(* IEC 61131-3 sources: com.logicals.lc3.webinar/logicals_Lib_Webinar/logicals_Webinar_Basic_Lib/logicals_Lib/src_FB_FBD/Convert, 5 files *)

(* ---- FB_lc_ByteNotNull_FBD.iecfbd ---- *)
NAMESPACE com.logicals.Basic.Convert
FUNCTION_BLOCK FB_lc_ByteNotNull_FBD
  {
    width := 170;
    minWidth := 160;
    maxWidth := 160;
    height := 198;
    minHeight := 198;
    maxHeight := 198;
  }

  VAR_INPUT
    vib_Byte9 : BYTE := 95;
    vib_Byte8 : BYTE := 95;
    vib_Byte7 : BYTE := 95;
    vib_Byte6 : BYTE := 95;
    vib_Byte5 : BYTE := 95;
    vib_Byte4 : BYTE := 95;
    vib_Byte3 : BYTE := 95;
    vib_Byte2 : BYTE := 95;
    vib_Byte1 : BYTE := 95;
    vib_Byte0 : BYTE := 95;
  END_VAR
  VAR_OUTPUT
    vob_Byte9 : BYTE := 95;
    vob_Byte8 : BYTE := 95;
    vob_Byte7 : BYTE := 95;
    vob_Byte6 : BYTE := 95;
    vob_Byte5 : BYTE := 95;
    vob_Byte4 : BYTE := 95;
    vob_Byte3 : BYTE := 95;
    vob_Byte2 : BYTE := 95;
    vob_Byte1 : BYTE := 95;
    vob_Byte0 : BYTE := 95;
  END_VAR

  (*

    // Network 1:
    EQ(IN1 := vib_Byte0, IN2 := 0, EQ => @C(161).EQ);
    SEL(G := @C(161).EQ, IN0 := vib_Byte0, IN1 := 95, SEL => vob_Byte0);

    // Network 2:
    EQ(IN1 := vib_Byte1, IN2 := 0, EQ => @C(160).EQ);
    SEL(G := @C(160).EQ, IN0 := vib_Byte1, IN1 := 95, SEL => vob_Byte1);

    // Network 3:
    EQ(IN1 := vib_Byte2, IN2 := 0, EQ => @C(164).EQ);
    SEL(G := @C(164).EQ, IN0 := vib_Byte2, IN1 := 95, SEL => vob_Byte2);

    // Network 4:
    EQ(IN1 := vib_Byte3, IN2 := 0, EQ => @C(162).EQ);
    SEL(G := @C(162).EQ, IN0 := vib_Byte3, IN1 := 95, SEL => vob_Byte3);

    // Network 5:
    EQ(IN1 := vib_Byte4, IN2 := 0, EQ => @C(166).EQ);
    SEL(G := @C(166).EQ, IN0 := vib_Byte4, IN1 := 95, SEL => vob_Byte4);

    // Network 6:
    EQ(IN1 := vib_Byte5, IN2 := 0, EQ => @C(169).EQ);
    SEL(G := @C(169).EQ, IN0 := vib_Byte5, IN1 := 95, SEL => vob_Byte5);

    // Network 7:
    EQ(IN1 := vib_Byte6, IN2 := 0, EQ => @C(165).EQ);
    SEL(G := @C(165).EQ, IN0 := vib_Byte6, IN1 := 95, SEL => vob_Byte6);

    // Network 8:
    EQ(IN1 := vib_Byte7, IN2 := 0, EQ => @C(168).EQ);
    SEL(G := @C(168).EQ, IN0 := vib_Byte7, IN1 := 95, SEL => vob_Byte7);

    // Network 9:
    EQ(IN1 := vib_Byte8, IN2 := 0, EQ => @C(163).EQ);
    SEL(G := @C(163).EQ, IN0 := vib_Byte8, IN1 := 95, SEL => vob_Byte8);

    // Network 10:
    EQ(IN1 := vib_Byte9, IN2 := 0, EQ => @C(167).EQ);
    SEL(G := @C(167).EQ, IN0 := vib_Byte9, IN1 := 95, SEL => vob_Byte9);

  *)

  @C(118) : @F(SEL), @R(810.0, 820.0, 120.0, 58.0), BYTE, @I(@N(G), @L(9.5)), @I(@N(IN0), @L(29.5)), @I(@N(IN1), @L(49.5)), @O(@N(SEL), @R(9.5));
  @C(150) : @F(SEL), @R(810.0, 730.0, 120.0, 58.0), BYTE, @I(@N(G), @L(9.5)), @I(@N(IN0), @L(29.5)), @I(@N(IN1), @L(49.5)), @O(@N(SEL), @R(9.5));
  @C(163) : @F(EQ), @R(540.0, 730.0, 40.0, 38.0), BYTE, @I(@N(IN1), @L(9.5)), @I(@N(IN2), @L(29.5)), @O(@N(EQ), @R(9.5));
  @C(167) : @F(EQ), @R(540.0, 820.0, 40.0, 38.0), BYTE, @I(@N(IN1), @L(9.5)), @I(@N(IN2), @L(29.5)), @O(@N(EQ), @R(9.5));
  @C(143) : @F(SEL), @R(810.0, 640.0, 120.0, 58.0), BYTE, @I(@N(G), @L(9.5)), @I(@N(IN0), @L(29.5)), @I(@N(IN1), @L(49.5)), @O(@N(SEL), @R(9.5));
  @C(168) : @F(EQ), @R(540.0, 640.0, 40.0, 38.0), BYTE, @I(@N(IN1), @L(9.5)), @I(@N(IN2), @L(29.5)), @O(@N(EQ), @R(9.5));
  @C(148) : @F(SEL), @R(810.0, 550.0, 120.0, 58.0), BYTE, @I(@N(G), @L(9.5)), @I(@N(IN0), @L(29.5)), @I(@N(IN1), @L(49.5)), @O(@N(SEL), @R(9.5));
  @C(165) : @F(EQ), @R(540.0, 550.0, 40.0, 38.0), BYTE, @I(@N(IN1), @L(9.5)), @I(@N(IN2), @L(29.5)), @O(@N(EQ), @R(9.5));
  @C(156) : @F(SEL), @R(810.0, 460.0, 120.0, 58.0), BYTE, @I(@N(G), @L(9.5)), @I(@N(IN0), @L(29.5)), @I(@N(IN1), @L(49.5)), @O(@N(SEL), @R(9.5));
  @C(169) : @F(EQ), @R(540.0, 460.0, 40.0, 38.0), BYTE, @I(@N(IN1), @L(9.5)), @I(@N(IN2), @L(29.5)), @O(@N(EQ), @R(9.5));
  @C(166) : @F(EQ), @R(540.0, 380.0, 40.0, 38.0), BYTE, @I(@N(IN1), @L(9.5)), @I(@N(IN2), @L(29.5)), @O(@N(EQ), @R(9.5));
  @C(115) : @F(SEL), @R(810.0, 380.0, 120.0, 58.0), BYTE, @I(@N(G), @L(9.5)), @I(@N(IN0), @L(29.5)), @I(@N(IN1), @L(49.5)), @O(@N(SEL), @R(9.5));
  @C(130) : @F(SEL), @R(810.0, 300.0, 120.0, 58.0), BYTE, @I(@N(G), @L(9.5)), @I(@N(IN0), @L(29.5)), @I(@N(IN1), @L(49.5)), @O(@N(SEL), @R(9.5));
  @C(162) : @F(EQ), @R(540.0, 300.0, 40.0, 38.0), BYTE, @I(@N(IN1), @L(9.5)), @I(@N(IN2), @L(29.5)), @O(@N(EQ), @R(9.5));
  @C(164) : @F(EQ), @R(540.0, 220.0, 40.0, 38.0), BYTE, @I(@N(IN1), @L(9.5)), @I(@N(IN2), @L(29.5)), @O(@N(EQ), @R(9.5));
  @C(105) : @F(SEL), @R(810.0, 220.0, 120.0, 58.0), BYTE, @I(@N(G), @L(9.5)), @I(@N(IN0), @L(29.5)), @I(@N(IN1), @L(49.5)), @O(@N(SEL), @R(9.5));
  @C(160) : @F(EQ), @R(540.0, 140.0, 40.0, 38.0), BYTE, @I(@N(IN1), @L(9.5)), @I(@N(IN2), @L(29.5)), @O(@N(EQ), @R(9.5));
  @C(121) : @F(SEL), @R(810.0, 140.0, 120.0, 58.0), BYTE, @I(@N(G), @L(9.5)), @I(@N(IN0), @L(29.5)), @I(@N(IN1), @L(49.5)), @O(@N(SEL), @R(9.5));
  @C(153) : @F(SEL), @R(810.0, 60.0, 120.0, 58.0), BYTE, @I(@N(G), @L(9.5)), @I(@N(IN0), @L(29.5)), @I(@N(IN1), @L(49.5)), @O(@N(SEL), @R(9.5));
  @C(161) : @F(EQ), @R(540.0, 60.0, 40.0, 38.0), BYTE, @I(@N(IN1), @L(9.5)), @I(@N(IN2), @L(29.5)), @O(@N(EQ), @R(9.5));
  @VF(117) : @E(vob_Byte9), @R(1460.0, 820.0, 100.0, 19.0);
  @VF(145) : @E(95), @R(680.0, 770.0, 60.0, 19.0), BYTE;
  @VF(119) : @E(95), @R(680.0, 860.0, 60.0, 19.0), BYTE;
  @VF(124) : @E(vib_Byte9), @R(680.0, 840.0, 100.0, 19.0);
  @VF(107) : @E(vib_Byte8), @R(680.0, 750.0, 100.0, 19.0);
  @VF(149) : @E(vob_Byte8), @R(1460.0, 730.0, 100.0, 19.0);
  @VF(141) : @E(0), @R(460.0, 840.0, 60.0, 19.0), BYTE;
  @VF(108) : @E(0), @R(460.0, 750.0, 60.0, 19.0), BYTE;
  @VF(159) : @E(95), @R(680.0, 680.0, 60.0, 19.0), BYTE;
  @VF(137) : @E(vib_Byte7), @R(680.0, 660.0, 100.0, 19.0);
  @VF(136) : @E(0), @R(460.0, 660.0, 60.0, 19.0), BYTE;
  @VF(142) : @E(vob_Byte7), @R(1460.0, 640.0, 100.0, 19.0);
  @VF(131) : @E(vib_Byte9), @R(280.0, 820.0, 100.0, 19.0);
  @VF(157) : @E(vib_Byte7), @R(280.0, 640.0, 100.0, 19.0);
  @VF(125) : @E(vib_Byte8), @R(280.0, 730.0, 100.0, 19.0);
  @VF(134) : @E(95), @R(680.0, 590.0, 60.0, 19.0), BYTE;
  @VF(109) : @E(vib_Byte6), @R(680.0, 570.0, 100.0, 19.0);
  @VF(127) : @E(0), @R(460.0, 570.0, 60.0, 19.0), BYTE;
  @VF(154) : @E(vib_Byte6), @R(280.0, 550.0, 100.0, 19.0);
  @VF(147) : @E(vob_Byte6), @R(1460.0, 550.0, 100.0, 19.0);
  @VF(101) : @E(95), @R(680.0, 500.0, 60.0, 19.0), BYTE;
  @VF(116) : @E(0), @R(460.0, 480.0, 60.0, 19.0), BYTE;
  @VF(113) : @E(vib_Byte5), @R(680.0, 480.0, 100.0, 19.0);
  @VF(155) : @E(vob_Byte5), @R(1460.0, 460.0, 100.0, 19.0);
  @VF(103) : @E(vib_Byte5), @R(280.0, 460.0, 100.0, 19.0);
  @VF(151) : @E(95), @R(680.0, 420.0, 60.0, 19.0), BYTE;
  @VF(139) : @E(0), @R(460.0, 400.0, 60.0, 19.0), BYTE;
  @VF(135) : @E(vib_Byte4), @R(680.0, 400.0, 100.0, 19.0);
  @VF(133) : @E(vib_Byte4), @R(280.0, 380.0, 100.0, 19.0);
  @VF(114) : @E(vob_Byte4), @R(1460.0, 380.0, 100.0, 19.0);
  @VF(126) : @E(95), @R(680.0, 340.0, 60.0, 19.0), BYTE;
  @VF(138) : @E(0), @R(460.0, 320.0, 60.0, 19.0), BYTE;
  @VF(146) : @E(vib_Byte3), @R(680.0, 320.0, 100.0, 19.0);
  @VF(129) : @E(vob_Byte3), @R(1460.0, 300.0, 100.0, 19.0);
  @VF(123) : @E(vib_Byte3), @R(280.0, 300.0, 100.0, 19.0);
  @VF(158) : @E(95), @R(680.0, 260.0, 60.0, 19.0), BYTE;
  @VF(102) : @E(0), @R(460.0, 240.0, 60.0, 19.0), BYTE;
  @VF(112) : @E(vib_Byte2), @R(680.0, 240.0, 100.0, 19.0);
  @VF(110) : @E(vib_Byte2), @R(280.0, 220.0, 100.0, 19.0);
  @VF(104) : @E(vob_Byte2), @R(1460.0, 220.0, 100.0, 19.0);
  @VF(122) : @E(95), @R(680.0, 180.0, 60.0, 19.0), BYTE;
  @VF(140) : @E(vib_Byte1), @R(280.0, 140.0, 100.0, 19.0);
  @VF(128) : @E(0), @R(460.0, 160.0, 60.0, 19.0), BYTE;
  @VF(144) : @E(vib_Byte1), @R(680.0, 160.0, 100.0, 19.0);
  @VF(120) : @E(vob_Byte1), @R(1460.0, 140.0, 100.0, 19.0);
  @VF(111) : @E(95), @R(680.0, 100.0, 60.0, 19.0), BYTE;
  @VF(100) : @E(vib_Byte0), @R(680.0, 80.0, 100.0, 19.0);
  @VF(106) : @E(0), @R(460.0, 80.0, 60.0, 19.0), BYTE;
  @VF(132) : @E(vib_Byte0), @R(280.0, 60.0, 100.0, 19.0);
  @VF(152) : @E(vob_Byte0), @R(1460.0, 60.0, 100.0, 19.0);

  @G(178) :
     @L(@C(118).SEL, @VF(117).i)
    ;
  @G(216) :
     @L(@VF(124).o, @C(118).IN0)
    ;
  @G(217) :
     @L(@VF(119).o, @C(118).IN1)
    ;
  @G(220) :
     @L(@VF(145).o, @C(150).IN1)
    ;
  @G(219) :
     @L(@VF(107).o, @C(150).IN0)
    ;
  @G(215) :
     @L(@C(167).EQ, @C(118).G)
    ;
  @G(173) :
     @L(@C(150).SEL, @VF(149).i)
    ;
  @G(218) :
     @L(@C(163).EQ, @C(150).G)
    ;
  @G(190) :
     @L(@VF(108).o, @C(163).IN2)
    ;
  @G(198) :
     @L(@VF(141).o, @C(167).IN2)
    ;
  @G(208) :
     @L(@VF(159).o, @C(143).IN1)
    ;
  @G(200) :
     @L(@VF(136).o, @C(168).IN2)
    ;
  @G(207) :
     @L(@VF(137).o, @C(143).IN0)
    ;
  @G(189) :
     @L(@VF(125).o, @C(163).IN1)
    ;
  @G(197) :
     @L(@VF(131).o, @C(167).IN1)
    ;
  @G(171) :
     @L(@C(143).SEL, @VF(142).i)
    ;
  @G(199) :
     @L(@VF(157).o, @C(168).IN1)
    ;
  @G(206) :
     @L(@C(168).EQ, @C(143).G)
    ;
  @G(214) :
     @L(@VF(134).o, @C(148).IN1)
    ;
  @G(194) :
     @L(@VF(127).o, @C(165).IN2)
    ;
  @G(213) :
     @L(@VF(109).o, @C(148).IN0)
    ;
  @G(172) :
     @L(@C(148).SEL, @VF(147).i)
    ;
  @G(193) :
     @L(@VF(154).o, @C(165).IN1)
    ;
  @G(212) :
     @L(@C(165).EQ, @C(148).G)
    ;
  @G(229) :
     @L(@VF(101).o, @C(156).IN1)
    ;
  @G(202) :
     @L(@VF(116).o, @C(169).IN2)
    ;
  @G(228) :
     @L(@VF(113).o, @C(156).IN0)
    ;
  @G(175) :
     @L(@C(156).SEL, @VF(155).i)
    ;
  @G(201) :
     @L(@VF(103).o, @C(169).IN1)
    ;
  @G(227) :
     @L(@C(169).EQ, @C(156).G)
    ;
  @G(211) :
     @L(@VF(151).o, @C(115).IN1)
    ;
  @G(196) :
     @L(@VF(139).o, @C(166).IN2)
    ;
  @G(210) :
     @L(@VF(135).o, @C(115).IN0)
    ;
  @G(177) :
     @L(@C(115).SEL, @VF(114).i)
    ;
  @G(195) :
     @L(@VF(133).o, @C(166).IN1)
    ;
  @G(209) :
     @L(@C(166).EQ, @C(115).G)
    ;
  @G(188) :
     @L(@VF(126).o, @C(130).IN1)
    ;
  @G(185) :
     @L(@VF(138).o, @C(162).IN2)
    ;
  @G(187) :
     @L(@VF(146).o, @C(130).IN0)
    ;
  @G(170) :
     @L(@C(130).SEL, @VF(129).i)
    ;
  @G(184) :
     @L(@VF(123).o, @C(162).IN1)
    ;
  @G(186) :
     @L(@C(162).EQ, @C(130).G)
    ;
  @G(205) :
     @L(@VF(158).o, @C(105).IN1)
    ;
  @G(192) :
     @L(@VF(102).o, @C(164).IN2)
    ;
  @G(204) :
     @L(@VF(112).o, @C(105).IN0)
    ;
  @G(176) :
     @L(@C(105).SEL, @VF(104).i)
    ;
  @G(191) :
     @L(@VF(110).o, @C(164).IN1)
    ;
  @G(203) :
     @L(@C(164).EQ, @C(105).G)
    ;
  @G(223) :
     @L(@VF(122).o, @C(121).IN1)
    ;
  @G(181) :
     @L(@VF(128).o, @C(160).IN2)
    ;
  @G(222) :
     @L(@VF(144).o, @C(121).IN0)
    ;
  @G(179) :
     @L(@C(121).SEL, @VF(120).i)
    ;
  @G(180) :
     @L(@VF(140).o, @C(160).IN1)
    ;
  @G(221) :
     @L(@C(160).EQ, @C(121).G)
    ;
  @G(226) :
     @L(@VF(111).o, @C(153).IN1)
    ;
  @G(183) :
     @L(@VF(106).o, @C(161).IN2)
    ;
  @G(225) :
     @L(@VF(100).o, @C(153).IN0)
    ;
  @G(174) :
     @L(@C(153).SEL, @VF(152).i)
    ;
  @G(182) :
     @L(@VF(132).o, @C(161).IN1)
    ;
  @G(224) :
     @L(@C(161).EQ, @C(153).G)
    ;
END_FUNCTION_BLOCK
END_NAMESPACE

(* ---- FB_lc_ChrToByte_FBD.iecfbd ---- *)
NAMESPACE com.logicals.Basic.Convert
FUNCTION_BLOCK FB_lc_ChrToByte_FBD
  {
    width := 200;
    height := 58;
    minWidth := 200;
    maxWidth := 200;
    minHeight := 58;
    maxHeight := 58;
  }

  VAR_INPUT
    vistr_Chr_127 : STRING[127] := '0';
  END_VAR
  VAR_OUTPUT
    vob_Out : BYTE;
  END_VAR

  (*

    // Network 1:
    FIND(IN1 := '!##%%&\()*+,-./0123456789:;<=>?@ABCDEFGHIJKLMNOPQRSTUVWXYZ[\]^_`abcdefghijklmnopqrstuvwxyz', IN2 := vistr_Chr_127, FIND => @C(110).FIND);
    EQ(IN1 := @C(110).FIND, IN2 := 1, EQ => @C(108).EQ);
    ADD(IN1 := @C(110).FIND, IN2 := 32, ADD => @C(109).ADD);
    SEL(G := @C(108).EQ, IN0 := @C(109).ADD, IN1 := 95, SEL => @C(107).SEL);
    TO_BYTE(IN := @C(107).SEL, TO_BYTE => vob_Out);

  *)

  @C(109) : @F(ADD), @R(1250.0, 300.0, 40.0, 38.0), USINT, @I(@N(IN1), @L(9.5)), @I(@N(IN2), @L(29.5)), @O(@N(ADD), @R(9.5));
  @C(106) : @F(TO_BYTE), @R(1520.0, 280.0, 80.0, 18.0), USINT, @I(@N(IN), @L(9.5)), @O(@N(TO_BYTE), @R(9.5));
  @C(107) : @F(SEL), @R(1370.0, 280.0, 120.0, 58.0), USINT, @I(@N(G), @L(9.5)), @I(@N(IN0), @L(29.5)), @I(@N(IN1), @L(49.5)), @O(@N(SEL), @R(9.5));
  @C(110) : @F(FIND), @R(1040.0, 200.0, 100.0, 38.0), USINT, @I(@N(IN1), @L(9.5)), @I(@N(IN2), @L(29.5)), @O(@N(FIND), @R(9.5));
  @C(108) : @F(EQ), @R(1250.0, 200.0, 40.0, 38.0), USINT, @I(@N(IN1), @L(9.5)), @I(@N(IN2), @L(29.5)), @O(@N(EQ), @R(9.5));
  @VF(100) : @E(95), @R(1310.0, 320.0, 40.0, 19.0), USINT;
  @VF(102) : @E(32), @R(1180.0, 320.0, 50.0, 19.0), USINT;
  @VF(105) : @E(vob_Out), @R(1680.0, 280.0, 190.0, 19.0);
  @VF(101) : @E(1), @R(1180.0, 220.0, 50.0, 19.0), USINT;
  @VF(104) : @E(vistr_Chr_127), @R(790.0, 220.0, 200.0, 19.0);
  @VF(103) : @E('!##%%&\()*+,-./0123456789:;<=>?@ABCDEFGHIJKLMNOPQRSTUVWXYZ[\]^_`abcdefghijklmnopqrstuvwxyz'), @R(20.0, 200.0, 970.0, 19.0);
  @CF(1) : @R(650.0, 60.0, 970.0, 99.0), @T("Wnadelt ein CHAR in BYTE um!"), @POU;
  @CP(117) : 1160.0, 209.5;

  @G(115) :
     @L(@VF(100).o, @C(107).IN1)
    ;
  @G(114) :
     @L(@C(109).ADD, @C(107).IN0)
    ;
  @G(119) :
     @L(@VF(102).o, @C(109).IN2)
    ;
  @G(111) :
     @L(@C(106).TO_BYTE, @VF(105).i)
    ;
  @G(112) :
     @L(@C(107).SEL, @C(106).IN)
    ;
  @G(118) :
     @L(@VF(101).o, @C(108).IN2)
    ;
  @G(113) :
     @L(@C(108).EQ, @C(107).G)
    ;
  @G(116) :
     @L(@C(110).FIND, @CP(117)),
     @L(@CP(117), @C(108).IN1),
     @L(@CP(117), @C(109).IN1)
    ;
  @G(121) :
     @L(@VF(104).o, @C(110).IN2)
    ;
  @G(120) :
     @L(@VF(103).o, @C(110).IN1)
    ;
END_FUNCTION_BLOCK
END_NAMESPACE

(* ---- FB_lc_RealTo12Byte_FBD.iecfbd ---- *)
NAMESPACE com.logicals.Basic.Convert
FUNCTION_BLOCK FB_lc_RealTo12Byte_FBD
  {
    instanceName := {visible};
    width := 180;
    height := 238;
    minWidth := 180;
    minHeight := 238;
    maxWidth := 180;
    maxHeight := 238;
    inputValueFieldAreaWidth := 110;
    outputValueFieldAreaWidth := 110;
  }

  VAR_INPUT
    vir_In : REAL := 0.0;
  END_VAR
  VAR_OUTPUT
    vob_Sign : BYTE := 43;
    vob_Mill : BYTE := 48;
    vob_00Thous : BYTE := 48;
    vob_0Thous : BYTE := 48;
    vob_Thous : BYTE := 48;
    vob_Hun : BYTE := 48;
    vob_Ten : BYTE := 48;
    vob_Single : BYTE := 48;
    vob_Dot : BYTE := 46;
    vob_DSing : BYTE := 48;
    vob_DTen : BYTE := 48;
    vob_DHund : BYTE := 48;
  END_VAR

  (*

    // Network 1:
    GE(IN1 := vir_In, IN2 := 0.0, GE => @C(188).GE);
    SEL(G := @C(188).GE, IN0 := 45, IN1 := 43, SEL => vob_Sign);
    ABS(IN := vir_In, ABS => @C(178).ABS);
    MUL(IN1 := @C(178).ABS, IN2 := 1000.0, MUL => @C(177).MUL);
    TO_DINT(IN := @C(177).MUL, TO_DINT => @C(112).TO_DINT);
    DIV(IN1 := @C(112).TO_DINT, IN2 := 1000000000, DIV => @C(101).DIV);
    ADD(IN1 := @C(101).DIV, IN2 := 48, ADD => @C(185).ADD);
    TO_BYTE(IN := @C(185).ADD, TO_BYTE => vob_Mill);
    MOD(IN1 := @C(112).TO_DINT, IN2 := 1000000000, MOD => @C(172).MOD);
    DIV(IN1 := @C(172).MOD, IN2 := 100000000, DIV => @C(110).DIV);
    ADD(IN1 := @C(110).DIV, IN2 := 48, ADD => @C(189).ADD);
    TO_BYTE(IN := @C(189).ADD, TO_BYTE => vob_00Thous);
    MOD(IN1 := @C(172).MOD, IN2 := 100000000, MOD => @C(183).MOD);
    DIV(IN1 := @C(183).MOD, IN2 := 10000000, DIV => @C(169).DIV);
    ADD(IN1 := @C(169).DIV, IN2 := 48, ADD => @C(168).ADD);
    TO_BYTE(IN := @C(168).ADD, TO_BYTE => vob_0Thous);
    MOD(IN1 := @C(183).MOD, IN2 := 10000000, MOD => @C(174).MOD);
    DIV(IN1 := @C(174).MOD, IN2 := 1000000, DIV => @C(173).DIV);
    ADD(IN1 := @C(173).DIV, IN2 := 48, ADD => @C(179).ADD);
    TO_BYTE(IN := @C(179).ADD, TO_BYTE => vob_Thous);
    MOD(IN1 := @C(174).MOD, IN2 := 1000000, MOD => @C(176).MOD);
    DIV(IN1 := @C(176).MOD, IN2 := 100000, DIV => @C(175).DIV);
    ADD(IN1 := @C(175).DIV, IN2 := 48, ADD => @C(182).ADD);
    TO_BYTE(IN := @C(182).ADD, TO_BYTE => vob_Hun);
    MOD(IN1 := @C(176).MOD, IN2 := 100000, MOD => );
    DIV(IN1 := @C(116).MOD, IN2 := 10000, DIV => @C(166).DIV);
    ADD(IN1 := @C(166).DIV, IN2 := 48, ADD => @C(170).ADD);
    TO_BYTE(IN := @C(170).ADD, TO_BYTE => vob_Ten);
    MOD(IN1 := @C(116).MOD, IN2 := 10000, MOD => @C(184).MOD);
    DIV(IN1 := @C(184).MOD, IN2 := 1000, DIV => @C(181).DIV);
    ADD(IN1 := @C(181).DIV, IN2 := 48, ADD => @C(180).ADD);
    TO_BYTE(IN := @C(180).ADD, TO_BYTE => vob_Single);
    MOD(IN1 := @C(184).MOD, IN2 := 1000, MOD => @C(187).MOD);
    DIV(IN1 := @C(187).MOD, IN2 := 100, DIV => @C(171).DIV);
    ADD(IN1 := @C(171).DIV, IN2 := 48, ADD => @C(167).ADD);
    TO_BYTE(IN := @C(167).ADD, TO_BYTE => vob_DSing);
    MOD(IN1 := @C(187).MOD, IN2 := 100, MOD => @C(186).MOD);
    DIV(IN1 := @C(186).MOD, IN2 := 10, DIV => @C(114).DIV);
    ADD(IN1 := @C(114).DIV, IN2 := 48, ADD => @C(108).ADD);
    TO_BYTE(IN := @C(108).ADD, TO_BYTE => vob_DTen);
    MOD(IN1 := @C(186).MOD, IN2 := 10, MOD => @C(190).MOD);
    ADD(IN1 := @C(190).MOD, IN2 := 48, ADD => @C(165).ADD);
    TO_BYTE(IN := @C(165).ADD, TO_BYTE => vob_DHund);

    // Network 2:
    vob_Dot := 46;

  *)

  @VF(128) : @E(vob_0Thous), @R(1790.0, 550.0, 110.0, 19.0);
  @VF(130) : @E(1000), @R(490.0, 930.0, 60.0, 19.0), DINT;
  @VF(131) : @E(vob_Ten), @R(1790.0, 840.0, 110.0, 19.0);
  @VF(133) : @E(1000.0), @R(160.0, 410.0, 90.0, 19.0), REAL;
  @VF(134) : @E(100), @R(700.0, 1030.0, 60.0, 19.0), DINT;
  @VF(135) : @E(48), @R(1410.0, 640.0, 40.0, 19.0), DINT;
  @VF(136) : @E(48), @R(550.0, 410.0, 40.0, 19.0), DINT;
  @VF(137) : @E(10000000), @R(700.0, 570.0, 90.0, 19.0), DINT;
  @VF(138) : @E(10), @R(950.0, 1110.0, 40.0, 19.0), DINT;
  @VF(139) : @E(48), @R(1410.0, 1110.0, 40.0, 19.0), DINT;
  @VF(140) : @E(10000), @R(170.0, 860.0, 110.0, 19.0), DINT;
  @VF(141) : @E(vob_Mill), @R(1790.0, 390.0, 110.0, 19.0);
  @VF(143) : @E(vob_DSing), @R(1790.0, 1010.0, 110.0, 19.0);
  @VF(145) : @E(0.0), @R(300.0, 290.0, 40.0, 19.0), REAL;
  @VF(146) : @E(48), @R(950.0, 1030.0, 40.0, 19.0), DINT;
  @VF(147) : @E(48), @R(540.0, 860.0, 40.0, 19.0), DINT;
  @VF(148) : @E(vob_DHund), @R(1790.0, 1170.0, 110.0, 19.0);
  @VF(150) : @E(48), @R(700.0, 930.0, 40.0, 19.0), DINT;
  @VF(151) : @E(vob_Thous), @R(1790.0, 620.0, 110.0, 19.0);
  @VF(153) : @E(vob_Hun), @R(1790.0, 690.0, 110.0, 19.0);
  @VF(155) : @E(vob_Sign), @R(1790.0, 270.0, 110.0, 19.0);
  @VF(157) : @E(48), @R(700.0, 500.0, 40.0, 19.0), DINT;
  @VF(158) : @E(vob_Single), @R(1790.0, 910.0, 110.0, 19.0);
  @VF(160) : @E(100000000), @R(420.0, 570.0, 100.0, 19.0), DINT;
  @VF(161) : @E(1000000000), @R(320.0, 410.0, 120.0, 19.0), DINT;
  @VF(162) : @E(48), @R(1410.0, 710.0, 40.0, 19.0), DINT;
  @VF(163) : @E(45), @R(410.0, 290.0, 40.0, 19.0), BYTE;
  @VF(164) : @E(43), @R(410.0, 310.0, 40.0, 19.0), BYTE;
  @VF(105) : @E(vir_In), @R(10.0, 270.0, 90.0, 19.0);
  @VF(118) : @E(48), @R(980.0, 570.0, 40.0, 19.0), DINT;
  @VF(119) : @E(vob_Dot), @R(1790.0, 950.0, 110.0, 19.0);
  @VF(120) : @E(46), @R(1660.0, 950.0, 40.0, 19.0), BYTE;
  @VF(121) : @E(100000), @R(1140.0, 710.0, 90.0, 19.0), DINT;
  @VF(122) : @E(1000000), @R(910.0, 640.0, 80.0, 19.0), DINT;
  @VF(123) : @E(vob_00Thous), @R(1790.0, 480.0, 110.0, 19.0);
  @VF(125) : @E(48), @R(1410.0, 1190.0, 40.0, 19.0), DINT;
  @VF(126) : @E(vob_DTen), @R(1790.0, 1090.0, 110.0, 19.0);
  @C(129) : @F(TO_BYTE), @R(1660.0, 550.0, 80.0, 18.0), DINT, @I(@N(IN), @L(9.5)), @O(@N(TO_BYTE), @R(9.5));
  @C(132) : @F(TO_BYTE), @R(1660.0, 840.0, 80.0, 18.0), DINT, @I(@N(IN), @L(9.5)), @O(@N(TO_BYTE), @R(9.5));
  @C(142) : @F(TO_BYTE), @R(1660.0, 390.0, 80.0, 18.0), DINT, @I(@N(IN), @L(9.5)), @O(@N(TO_BYTE), @R(9.5));
  @C(144) : @F(TO_BYTE), @R(1660.0, 1010.0, 80.0, 18.0), DINT, @I(@N(IN), @L(9.5)), @O(@N(TO_BYTE), @R(9.5));
  @C(149) : @F(TO_BYTE), @R(1660.0, 1170.0, 80.0, 18.0), DINT, @I(@N(IN), @L(9.5)), @O(@N(TO_BYTE), @R(9.5));
  @C(152) : @F(TO_BYTE), @R(1660.0, 620.0, 80.0, 18.0), DINT, @I(@N(IN), @L(9.5)), @O(@N(TO_BYTE), @R(9.5));
  @C(154) : @F(TO_BYTE), @R(1660.0, 690.0, 80.0, 18.0), DINT, @I(@N(IN), @L(9.5)), @O(@N(TO_BYTE), @R(9.5));
  @C(156) : @F(SEL), @R(470.0, 270.0, 120.0, 58.0), BYTE, @I(@N(G), @L(9.5)), @I(@N(IN0), @L(29.5)), @I(@N(IN1), @L(49.5)), @O(@N(SEL), @R(9.5));
  @C(159) : @F(TO_BYTE), @R(1660.0, 910.0, 80.0, 18.0), DINT, @I(@N(IN), @L(9.5)), @O(@N(TO_BYTE), @R(9.5));
  @C(101) : @F(DIV), @R(500.0, 390.0, 40.0, 38.0), DINT, @I(@N(IN1), @L(9.5)), @I(@N(IN2), @L(29.5)), @O(@N(DIV), @R(9.5));
  @C(165) : @F(ADD), @R(1480.0, 1170.0, 40.0, 38.0), DINT, @I(@N(IN1), @L(9.5)), @I(@N(IN2), @L(29.5)), @O(@N(ADD), @R(9.5));
  @C(166) : @F(DIV), @R(490.0, 840.0, 40.0, 38.0), DINT, @I(@N(IN1), @L(9.5)), @I(@N(IN2), @L(29.5)), @O(@N(DIV), @R(9.5));
  @C(167) : @F(ADD), @R(1070.0, 1010.0, 40.0, 38.0), DINT, @I(@N(IN1), @L(9.5)), @I(@N(IN2), @L(29.5)), @O(@N(ADD), @R(9.5));
  @C(168) : @F(ADD), @R(1060.0, 550.0, 40.0, 38.0), DINT, @I(@N(IN1), @L(9.5)), @I(@N(IN2), @L(29.5)), @O(@N(ADD), @R(9.5));
  @C(169) : @F(DIV), @R(840.0, 550.0, 40.0, 38.0), DINT, @I(@N(IN1), @L(9.5)), @I(@N(IN2), @L(29.5)), @O(@N(DIV), @R(9.5));
  @C(170) : @F(ADD), @R(620.0, 840.0, 40.0, 38.0), DINT, @I(@N(IN1), @L(9.5)), @I(@N(IN2), @L(29.5)), @O(@N(ADD), @R(9.5));
  @C(171) : @F(DIV), @R(860.0, 1010.0, 40.0, 38.0), DINT, @I(@N(IN1), @L(9.5)), @I(@N(IN2), @L(29.5)), @O(@N(DIV), @R(9.5));
  @C(172) : @F(MOD), @R(500.0, 480.0, 60.0, 38.0), DINT, @I(@N(IN1), @L(9.5)), @I(@N(IN2), @L(29.5)), @O(@N(MOD), @R(9.5));
  @C(108) : @F(ADD), @R(1480.0, 1090.0, 40.0, 38.0), DINT, @I(@N(IN1), @L(9.5)), @I(@N(IN2), @L(29.5)), @O(@N(ADD), @R(9.5));
  @C(173) : @F(DIV), @R(1060.0, 620.0, 40.0, 38.0), DINT, @I(@N(IN1), @L(9.5)), @I(@N(IN2), @L(29.5)), @O(@N(DIV), @R(9.5));
  @C(110) : @F(DIV), @R(630.0, 480.0, 40.0, 38.0), DINT, @I(@N(IN1), @L(9.5)), @I(@N(IN2), @L(29.5)), @O(@N(DIV), @R(9.5));
  @C(174) : @F(MOD), @R(840.0, 620.0, 60.0, 38.0), DINT, @I(@N(IN1), @L(9.5)), @I(@N(IN2), @L(29.5)), @O(@N(MOD), @R(9.5));
  @C(175) : @F(DIV), @R(1330.0, 690.0, 40.0, 38.0), DINT, @I(@N(IN1), @L(9.5)), @I(@N(IN2), @L(29.5)), @O(@N(DIV), @R(9.5));
  @C(112) : @F(TO_DINT), @R(320.0, 390.0, 80.0, 18.0), REAL, @I(@N(IN), @L(9.5)), @O(@N(TO_DINT), @R(9.5));
  @C(176) : @F(MOD), @R(1060.0, 690.0, 60.0, 38.0), DINT, @I(@N(IN1), @L(9.5)), @I(@N(IN2), @L(29.5)), @O(@N(MOD), @R(9.5));
  @C(177) : @F(MUL), @R(270.0, 390.0, 40.0, 38.0), REAL, @I(@N(IN1), @L(9.5)), @I(@N(IN2), @L(29.5)), @O(@N(MUL), @R(9.5));
  @C(178) : @F(ABS), @R(190.0, 390.0, 60.0, 18.0), REAL, @I(@N(IN), @L(9.5)), @O(@N(ABS), @R(9.5));
  @C(114) : @F(DIV), @R(1070.0, 1090.0, 40.0, 38.0), DINT, @I(@N(IN1), @L(9.5)), @I(@N(IN2), @L(29.5)), @O(@N(DIV), @R(9.5));
  @C(179) : @F(ADD), @R(1480.0, 620.0, 40.0, 38.0), DINT, @I(@N(IN1), @L(9.5)), @I(@N(IN2), @L(29.5)), @O(@N(ADD), @R(9.5));
  @C(180) : @F(ADD), @R(860.0, 910.0, 40.0, 38.0), DINT, @I(@N(IN1), @L(9.5)), @I(@N(IN2), @L(29.5)), @O(@N(ADD), @R(9.5));
  @C(116) : @F(MOD), @R(1310.0, 760.0, 60.0, 38.0), DINT, @I(@N(IN1), @L(9.5)), @I(@N(IN2), @L(29.5)), @O(@N(MOD), @R(9.5));
  @C(181) : @F(DIV), @R(620.0, 910.0, 40.0, 38.0), DINT, @I(@N(IN1), @L(9.5)), @I(@N(IN2), @L(29.5)), @O(@N(DIV), @R(9.5));
  @C(182) : @F(ADD), @R(1480.0, 690.0, 40.0, 38.0), DINT, @I(@N(IN1), @L(9.5)), @I(@N(IN2), @L(29.5)), @O(@N(ADD), @R(9.5));
  @C(183) : @F(MOD), @R(630.0, 550.0, 60.0, 38.0), DINT, @I(@N(IN1), @L(9.5)), @I(@N(IN2), @L(29.5)), @O(@N(MOD), @R(9.5));
  @C(184) : @F(MOD), @R(420.0, 910.0, 60.0, 38.0), DINT, @I(@N(IN1), @L(9.5)), @I(@N(IN2), @L(29.5)), @O(@N(MOD), @R(9.5));
  @C(185) : @F(ADD), @R(630.0, 390.0, 40.0, 38.0), DINT, @I(@N(IN1), @L(9.5)), @I(@N(IN2), @L(29.5)), @O(@N(ADD), @R(9.5));
  @C(186) : @F(MOD), @R(860.0, 1090.0, 60.0, 38.0), DINT, @I(@N(IN1), @L(9.5)), @I(@N(IN2), @L(29.5)), @O(@N(MOD), @R(9.5));
  @C(187) : @F(MOD), @R(620.0, 1010.0, 60.0, 38.0), DINT, @I(@N(IN1), @L(9.5)), @I(@N(IN2), @L(29.5)), @O(@N(MOD), @R(9.5));
  @C(188) : @F(GE), @R(360.0, 270.0, 40.0, 38.0), REAL, @I(@N(IN1), @L(9.5)), @I(@N(IN2), @L(29.5)), @O(@N(GE), @R(9.5));
  @C(124) : @F(TO_BYTE), @R(1660.0, 480.0, 80.0, 18.0), DINT, @I(@N(IN), @L(9.5)), @O(@N(TO_BYTE), @R(9.5));
  @C(189) : @F(ADD), @R(840.0, 480.0, 40.0, 38.0), DINT, @I(@N(IN1), @L(9.5)), @I(@N(IN2), @L(29.5)), @O(@N(ADD), @R(9.5));
  @C(190) : @F(MOD), @R(1070.0, 1170.0, 60.0, 38.0), DINT, @I(@N(IN1), @L(9.5)), @I(@N(IN2), @L(29.5)), @O(@N(MOD), @R(9.5));
  @C(127) : @F(TO_BYTE), @R(1660.0, 1090.0, 80.0, 18.0), DINT, @I(@N(IN), @L(9.5)), @O(@N(TO_BYTE), @R(9.5));
  @CONN(115) : @IT(Rest), @R(1660.0, 760.0, 60.0, 19.0), DINT;
  @CONT(117) : @IT(Rest), @CONN(115), @R(121.0, 840.0, 157.0, 19.0), DINT;
  @CF(103) : @R(360.0, 95.0, 578.0, 63.0), @T("Real Value to 12 Character ASCII Byte Value$R$N$R$NRange: +/-0.001 $a0to $a0+/-2 147 483.000$R$N"), @POU;
  @CF(106) : @R(1560.0, 950.0, 87.0, 18.0), @T("Dot $".$""), @POU;
  @OLT(113) : @R(1130.0, 1040.0, 66.0, 19.0), @S(114,DIV);
  @OLT(104) : @R(170.0, 230.0, 108.0, 18.0), @S(105);
  @OLT(107) : @R(1540.0, 1030.0, 66.0, 19.0), @S(108,ADD);
  @OLT(109) : @R(700.0, 450.0, 40.0, 19.0), @S(110,DIV);
  @CF(20) : @R(1550.0, 230.0, 200.0, 29.0), @T("Sign / Vorzeichen"), @POU;
  @CF(21) : @R(500.0, 360.0, 60.0, 19.0), @T("DIV1"), @POU;
  @CF(22) : @R(630.0, 360.0, 60.0, 19.0), @T("ADD1"), @POU;
  @CF(23) : @R(630.0, 450.0, 60.0, 19.0), @T("DIV1"), @POU;
  @CF(24) : @R(500.0, 450.0, 60.0, 19.0), @T("MOD1"), @POU;
  @CF(25) : @R(840.0, 450.0, 60.0, 19.0), @T("ADD2"), @POU;
  @CF(26) : @R(630.0, 520.0, 60.0, 19.0), @T("MOD2"), @POU;
  @CF(27) : @R(840.0, 520.0, 60.0, 19.0), @T("DIV2"), @POU;
  @CF(28) : @R(1060.0, 520.0, 60.0, 19.0), @T("ADD3"), @POU;
  @CF(29) : @R(840.0, 590.0, 60.0, 19.0), @T("MOD3"), @POU;
  @CF(30) : @R(1060.0, 590.0, 60.0, 19.0), @T("DIV3"), @POU;
  @CF(31) : @R(1480.0, 590.0, 60.0, 19.0), @T("ADD4"), @POU;
  @CF(32) : @R(1060.0, 660.0, 60.0, 19.0), @T("MOD4"), @POU;
  @CF(33) : @R(1480.0, 660.0, 60.0, 19.0), @T("ADD5"), @POU;
  @CF(34) : @R(1330.0, 660.0, 60.0, 19.0), @T("DIV4"), @POU;
  @CF(35) : @R(1310.0, 730.0, 60.0, 19.0), @T("MOD5"), @POU;
  @CF(36) : @R(490.0, 810.0, 60.0, 19.0), @T("DIV5"), @POU;
  @CF(37) : @R(620.0, 810.0, 60.0, 19.0), @T("ADD6"), @POU;
  @CF(38) : @R(420.0, 880.0, 60.0, 19.0), @T("MOD6"), @POU;
  @CF(39) : @R(620.0, 880.0, 60.0, 19.0), @T("DIV6"), @POU;
  @CF(40) : @R(860.0, 880.0, 60.0, 19.0), @T("ADD7"), @POU;
  @CF(41) : @R(620.0, 980.0, 60.0, 19.0), @T("MOD7"), @POU;
  @CF(42) : @R(860.0, 980.0, 60.0, 19.0), @T("DIV7"), @POU;
  @CF(43) : @R(1070.0, 980.0, 60.0, 19.0), @T("ADD8"), @POU;
  @CF(44) : @R(860.0, 1060.0, 60.0, 19.0), @T("MOD8"), @POU;
  @CF(45) : @R(1070.0, 1060.0, 60.0, 19.0), @T("DIV8"), @POU;
  @CF(46) : @R(1480.0, 1060.0, 60.0, 19.0), @T("ADD9"), @POU;
  @CF(47) : @R(1070.0, 1140.0, 60.0, 19.0), @T("MOD9"), @POU;
  @CF(48) : @R(1480.0, 1140.0, 60.0, 19.0), @T("ADD10"), @POU;
  @OLT(49) : @R(1790.0, 370.0, 80.0, 19.0), @S(141);
  @OLT(50) : @R(1790.0, 460.0, 80.0, 19.0), @S(123);
  @OLT(51) : @R(1790.0, 530.0, 80.0, 19.0), @S(128);
  @OLT(52) : @R(1790.0, 600.0, 80.0, 19.0), @S(151);
  @OLT(53) : @R(1790.0, 670.0, 80.0, 19.0), @S(153);
  @OLT(54) : @R(1790.0, 820.0, 80.0, 19.0), @S(131);
  @OLT(55) : @R(1790.0, 890.0, 80.0, 19.0), @S(158);
  @OLT(56) : @R(1790.0, 930.0, 80.0, 19.0), @S(119);
  @OLT(57) : @R(1790.0, 990.0, 80.0, 19.0), @S(143);
  @OLT(58) : @R(1790.0, 1070.0, 80.0, 19.0), @S(126);
  @OLT(59) : @R(1790.0, 1150.0, 80.0, 19.0), @S(148);
  @OLT(60) : @R(270.0, 350.0, 130.0, 19.0), @S(112,TO_DINT);
  @OLT(61) : @R(710.0, 360.0, 40.0, 19.0), @S(185,ADD);
  @OLT(62) : @R(560.0, 810.0, 50.0, 19.0), @S(166,DIV);
  @OLT(63) : @R(710.0, 880.0, 40.0, 19.0), @S(181,DIV);
  @OLT(64) : @R(1410.0, 780.0, 80.0, 19.0), @S(116,MOD);
  @OLT(65) : @R(1150.0, 660.0, 80.0, 19.0), @S(176,MOD);
  @OLT(66) : @R(1140.0, 590.0, 80.0, 19.0), @S(173,DIV);
  @OLT(67) : @R(910.0, 590.0, 80.0, 19.0), @S(174,MOD);
  @OLT(68) : @R(1410.0, 670.0, 40.0, 19.0), @S(175,DIV);
  @OLT(69) : @R(920.0, 520.0, 80.0, 19.0), @S(169,DIV);
  @OLT(70) : @R(700.0, 520.0, 130.0, 19.0), @S(183,MOD);
  @OLT(71) : @R(630.0, 310.0, 80.0, 19.0), @S(101,DIV);
  @OLT(72) : @R(380.0, 530.0, 120.0, 19.0), @S(172,MOD);
  @CP(221) : 410.0, 849.5;
  @CP(223) : 390.0, 869.5;
  @CP(245) : 620.0, 489.5;
  @CP(256) : 170.0, 279.5;
  @CP(1) : 1279.5, 699.5;
  @CP(2) : 1259.5, 719.5;
  @CP(4) : 1029.5, 629.5;
  @CP(6) : 1009.5, 649.5;
  @CP(7) : 819.5, 559.5;
  @CP(9) : 799.5, 579.5;
  @CP(11) : 579.5, 579.5;
  @CP(12) : 1039.5, 1099.5;
  @CP(13) : 1009.5, 1119.5;
  @CP(14) : 829.5, 1019.5;
  @CP(15) : 799.5, 1039.5;
  @CP(16) : 479.5, 399.5;
  @CP(17) : 459.5, 419.5;
  @CP(18) : 599.5, 919.5;
  @CP(19) : 579.5, 939.5;

  @G(191) :
     @L(@C(129).TO_BYTE, @VF(128).i)
    ;
  @G(192) :
     @L(@C(132).TO_BYTE, @VF(131).i)
    ;
  @G(193) :
     @L(@C(142).TO_BYTE, @VF(141).i)
    ;
  @G(194) :
     @L(@C(144).TO_BYTE, @VF(143).i)
    ;
  @G(195) :
     @L(@C(149).TO_BYTE, @VF(148).i)
    ;
  @G(196) :
     @L(@C(152).TO_BYTE, @VF(151).i)
    ;
  @G(197) :
     @L(@C(154).TO_BYTE, @VF(153).i)
    ;
  @G(198) :
     @L(@C(156).SEL, @VF(155).i)
    ;
  @G(199) :
     @L(@C(159).TO_BYTE, @VF(158).i)
    ;
  @G(200) :
     @L(@VF(120).o, @VF(119).i)
    ;
  @G(201) :
     @L(@C(124).TO_BYTE, @VF(123).i)
    ;
  @G(202) :
     @L(@C(127).TO_BYTE, @VF(126).i)
    ;
  @G(203) :
     @L(@C(168).ADD, @C(129).IN)
    ;
  @G(204) :
     @L(@C(170).ADD, @C(132).IN)
    ;
  @G(205) :
     @L(@C(185).ADD, @C(142).IN)
    ;
  @G(206) :
     @L(@C(167).ADD, @C(144).IN)
    ;
  @G(207) :
     @L(@C(165).ADD, @C(149).IN)
    ;
  @G(208) :
     @L(@C(179).ADD, @C(152).IN)
    ;
  @G(209) :
     @L(@C(182).ADD, @C(154).IN)
    ;
  @G(210) :
     @L(@C(188).GE, @C(156).G)
    ;
  @G(211) :
     @L(@VF(163).o, @C(156).IN0)
    ;
  @G(212) :
     @L(@VF(164).o, @C(156).IN1)
    ;
  @G(213) :
     @L(@C(180).ADD, @C(159).IN)
    ;
  @G(214) :
     @L(@C(112).TO_DINT, @CP(16)),
     @L(@CP(16), @C(101).IN1),
     @L(@CP(16), @C(172).IN1)
    ;
  @G(216) :
     @L(@VF(161).o, @CP(17)),
     @L(@CP(17), @C(101).IN2),
     @L(@CP(17), @C(172).IN2)
    ;
  @G(218) :
     @L(@C(190).MOD, @C(165).IN1)
    ;
  @G(219) :
     @L(@VF(125).o, @C(165).IN2)
    ;
  @G(220) :
     @L(@CONT(117).o, @CP(221)),
     @L(@CP(221), @C(166).IN1),
     @L(@CP(221), @C(184).IN1)
    ;
  @G(222) :
     @L(@VF(140).o, @CP(223)),
     @L(@CP(223), @C(166).IN2),
     @L(@CP(223), @C(184).IN2)
    ;
  @G(224) :
     @L(@C(171).DIV, @C(167).IN1)
    ;
  @G(225) :
     @L(@VF(146).o, @C(167).IN2)
    ;
  @G(226) :
     @L(@C(169).DIV, @C(168).IN1)
    ;
  @G(227) :
     @L(@VF(118).o, @C(168).IN2)
    ;
  @G(228) :
     @L(@C(183).MOD, @CP(7)),
     @L(@CP(7), @C(169).IN1),
     @L(@CP(7), @C(174).IN1)
    ;
  @G(232) :
     @L(@C(166).DIV, @C(170).IN1)
    ;
  @G(233) :
     @L(@VF(147).o, @C(170).IN2)
    ;
  @G(234) :
     @L(@C(187).MOD, @CP(14)),
     @L(@CP(14), @C(171).IN1),
     @L(@CP(14), @C(186).IN1)
    ;
  @G(236) :
     @L(@VF(134).o, @CP(15)),
     @L(@CP(15), @C(171).IN2),
     @L(@CP(15), @C(186).IN2)
    ;
  @G(238) :
     @L(@C(114).DIV, @C(108).IN1)
    ;
  @G(239) :
     @L(@VF(139).o, @C(108).IN2)
    ;
  @G(244) :
     @L(@C(172).MOD, @CP(245)),
     @L(@CP(245), @C(110).IN1),
     @L(@CP(245), @C(183).IN1)
    ;
  @G(248) :
     @L(@C(176).MOD, @CP(1)),
     @L(@CP(1), @C(175).IN1),
     @L(@CP(1), @C(116).IN1)
    ;
  @G(250) :
     @L(@VF(121).o, @CP(2)),
     @L(@CP(2), @C(175).IN2),
     @L(@CP(2), @C(116).IN2)
    ;
  @G(252) :
     @L(@C(177).MUL, @C(112).IN)
    ;
  @G(253) :
     @L(@C(178).ABS, @C(177).IN1)
    ;
  @G(254) :
     @L(@VF(133).o, @C(177).IN2)
    ;
  @G(255) :
     @L(@VF(105).o, @CP(256)),
     @L(@CP(256), @C(178).IN),
     @L(@CP(256), @C(188).IN1)
    ;
  @G(257) :
     @L(@C(186).MOD, @CP(12)),
     @L(@CP(12), @C(114).IN1),
     @L(@CP(12), @C(190).IN1)
    ;
  @G(259) :
     @L(@VF(138).o, @CP(13)),
     @L(@CP(13), @C(114).IN2),
     @L(@CP(13), @C(190).IN2)
    ;
  @G(261) :
     @L(@C(173).DIV, @C(179).IN1)
    ;
  @G(262) :
     @L(@VF(135).o, @C(179).IN2)
    ;
  @G(263) :
     @L(@C(181).DIV, @C(180).IN1)
    ;
  @G(264) :
     @L(@VF(150).o, @C(180).IN2)
    ;
  @G(265) :
     @L(@C(184).MOD, @CP(18)),
     @L(@CP(18), @C(181).IN1),
     @L(@CP(18), @C(187).IN1)
    ;
  @G(267) :
     @L(@VF(130).o, @CP(19)),
     @L(@CP(19), @C(181).IN2),
     @L(@CP(19), @C(187).IN2)
    ;
  @G(269) :
     @L(@C(175).DIV, @C(182).IN1)
    ;
  @G(270) :
     @L(@VF(162).o, @C(182).IN2)
    ;
  @G(271) :
     @L(@C(101).DIV, @C(185).IN1)
    ;
  @G(272) :
     @L(@VF(136).o, @C(185).IN2)
    ;
  @G(273) :
     @L(@VF(145).o, @C(188).IN2)
    ;
  @G(274) :
     @L(@C(189).ADD, @C(124).IN)
    ;
  @G(275) :
     @L(@C(110).DIV, @C(189).IN1)
    ;
  @G(276) :
     @L(@VF(157).o, @C(189).IN2)
    ;
  @G(277) :
     @L(@C(108).ADD, @C(127).IN)
    ;
  @G(278) :
     @L(@C(116).MOD, @CONN(115).i)
    ;
  @G(3) :
     @L(@C(174).MOD, @CP(4)),
     @L(@CP(4), @C(173).IN1),
     @L(@CP(4), @C(176).IN1)
    ;
  @G(5) :
     @L(@VF(122).o, @CP(6)),
     @L(@CP(6), @C(173).IN2),
     @L(@CP(6), @C(176).IN2)
    ;
  @G(8) :
     @L(@VF(137).o, @CP(9)),
     @L(@CP(9), @C(169).IN2),
     @L(@CP(9), @C(174).IN2)
    ;
  @G(10) :
     @L(@VF(160).o, @CP(11)),
     @L(@CP(11), @C(183).IN2),
     @L(@CP(11), @C(110).IN2)
    ;
END_FUNCTION_BLOCK
END_NAMESPACE

(* ---- FB_lc_StrTo10Byte_FBD.iecfbd ---- *)
NAMESPACE com.logicals.Basic.Convert
FUNCTION_BLOCK FB_lc_StrTo10Byte_FBD
  {
    altName := "StrToBy";
    width := 180;
    minWidth := 180;
    minHeight := 238;
    maxWidth := 180;
    maxHeight := 238;
    pageSize := "1340x950";
    inputValueFieldAreaWidth := 160;
    outputValueFieldAreaWidth := 160;
    height := 238;
  }

  VAR
    FB_lc_ChrToByte : FB_lc_ChrToByte_FBD;
    FB_lc_ChrToByte1 : FB_lc_ChrToByte_FBD;
    FB_lc_ChrToByte2 : FB_lc_ChrToByte_FBD;
    FB_lc_ChrToByte3 : FB_lc_ChrToByte_FBD;
    FB_lc_ChrToByte4 : FB_lc_ChrToByte_FBD;
    FB_lc_ChrToByte5 : FB_lc_ChrToByte_FBD;
    FB_lc_ChrToByte6 : FB_lc_ChrToByte_FBD;
    FB_lc_ChrToByte7 : FB_lc_ChrToByte_FBD;
    FB_lc_ChrToByte8 : FB_lc_ChrToByte_FBD;
    FB_lc_ChrToByte9 : FB_lc_ChrToByte_FBD;
  END_VAR
  VAR_INPUT
    vistr_In_127 : STRING[127];
  END_VAR
  VAR_OUTPUT
    vob_Byte0 : BYTE;
    vob_Byte1 : BYTE;
    vob_Byte2 : BYTE;
    vob_Byte3 : BYTE;
    vob_Byte4 : BYTE;
    vob_Byte5 : BYTE;
    vob_Byte6 : BYTE;
    vob_Byte7 : BYTE;
    vob_Byte8 : BYTE;
    vob_Byte9 : BYTE;
  END_VAR

  (*

    // Network 1:
    TO_INT(IN := 1, TO_INT => @C(148).TO_INT);
    TO_INT(IN := 1, TO_INT => @C(160).TO_INT);
    MID(IN := vistr_In_127, L := @C(148).TO_INT, P := @C(160).TO_INT, MID => @C(153).MID);
    FB_lc_ChrToByte2(vistr_Chr_127 := @C(153).MID, vob_Out => vob_Byte0);
    TO_INT(IN := 1, TO_INT => @C(142).TO_INT);
    TO_INT(IN := 2, TO_INT => @C(143).TO_INT);
    MID(IN := vistr_In_127, L := @C(142).TO_INT, P := @C(143).TO_INT, MID => @C(141).MID);
    FB_lc_ChrToByte1(vistr_Chr_127 := @C(141).MID, vob_Out => vob_Byte1);
    TO_INT(IN := 1, TO_INT => @C(169).TO_INT);
    TO_INT(IN := 3, TO_INT => @C(159).TO_INT);
    MID(IN := vistr_In_127, L := @C(169).TO_INT, P := @C(159).TO_INT, MID => @C(144).MID);
    FB_lc_ChrToByte(vistr_Chr_127 := @C(144).MID, vob_Out => vob_Byte2);
    TO_INT(IN := 1, TO_INT => @C(168).TO_INT);
    TO_INT(IN := 4, TO_INT => @C(170).TO_INT);
    MID(IN := vistr_In_127, L := @C(168).TO_INT, P := @C(170).TO_INT, MID => @C(167).MID);
    FB_lc_ChrToByte3(vistr_Chr_127 := @C(167).MID, vob_Out => vob_Byte3);
    TO_INT(IN := 1, TO_INT => @C(149).TO_INT);
    TO_INT(IN := 5, TO_INT => @C(157).TO_INT);
    MID(IN := vistr_In_127, L := @C(149).TO_INT, P := @C(157).TO_INT, MID => @C(156).MID);
    FB_lc_ChrToByte4(vistr_Chr_127 := @C(156).MID, vob_Out => vob_Byte4);
    TO_INT(IN := 1, TO_INT => @C(154).TO_INT);
    TO_INT(IN := 6, TO_INT => @C(158).TO_INT);
    MID(IN := vistr_In_127, L := @C(154).TO_INT, P := @C(158).TO_INT, MID => @C(155).MID);
    FB_lc_ChrToByte5(vistr_Chr_127 := @C(155).MID, vob_Out => vob_Byte5);
    TO_INT(IN := 1, TO_INT => @C(151).TO_INT);
    TO_INT(IN := 7, TO_INT => @C(152).TO_INT);
    MID(IN := vistr_In_127, L := @C(151).TO_INT, P := @C(152).TO_INT, MID => @C(150).MID);
    FB_lc_ChrToByte6(vistr_Chr_127 := @C(150).MID, vob_Out => vob_Byte6);
    TO_INT(IN := 1, TO_INT => @C(165).TO_INT);
    TO_INT(IN := 8, TO_INT => @C(166).TO_INT);
    MID(IN := vistr_In_127, L := @C(165).TO_INT, P := @C(166).TO_INT, MID => @C(164).MID);
    FB_lc_ChrToByte7(vistr_Chr_127 := @C(164).MID, vob_Out => vob_Byte7);
    TO_INT(IN := 1, TO_INT => @C(146).TO_INT);
    TO_INT(IN := 9, TO_INT => @C(147).TO_INT);
    MID(IN := vistr_In_127, L := @C(146).TO_INT, P := @C(147).TO_INT, MID => @C(145).MID);
    FB_lc_ChrToByte8(vistr_Chr_127 := @C(145).MID, vob_Out => vob_Byte8);
    TO_INT(IN := 1, TO_INT => @C(162).TO_INT);
    TO_INT(IN := 10, TO_INT => @C(163).TO_INT);
    MID(IN := vistr_In_127, L := @C(162).TO_INT, P := @C(163).TO_INT, MID => @C(161).MID);
    FB_lc_ChrToByte9(vistr_Chr_127 := @C(161).MID, vob_Out => vob_Byte9);

  *)

  @VF(129) : @E(1), @R(320.0, 690.0, 40.0, 19.0), BOOL;
  @VF(130) : @E(2), @R(320.0, 150.0, 40.0, 19.0), BYTE;
  @VF(131) : @E(8), @R(320.0, 710.0, 40.0, 19.0), BYTE;
  @VF(132) : @E(vistr_In_127), @R(0.0, 20.0, 190.0, 19.0);
  @VF(133) : @E(9), @R(320.0, 800.0, 40.0, 19.0), BYTE;
  @VF(134) : @E(1), @R(320.0, 320.0, 40.0, 19.0), BOOL;
  @VF(135) : @E(10), @R(320.0, 890.0, 40.0, 19.0), BYTE;
  @VF(136) : @E(1), @R(320.0, 600.0, 40.0, 19.0), BOOL;
  @VF(137) : @E(5), @R(320.0, 430.0, 40.0, 19.0), BYTE;
  @VF(138) : @E(6), @R(320.0, 520.0, 40.0, 19.0), BYTE;
  @VF(139) : @E(vob_Byte8), @R(1190.0, 760.0, 110.0, 19.0);
  @VF(100) : @E(1), @R(320.0, 500.0, 40.0, 19.0), BOOL;
  @VF(101) : @E(vob_Byte2), @R(1190.0, 210.0, 110.0, 19.0);
  @VF(103) : @E(vob_Byte5), @R(1190.0, 480.0, 110.0, 19.0);
  @VF(105) : @E(7), @R(320.0, 620.0, 40.0, 19.0), BYTE;
  @VF(106) : @E(1), @R(320.0, 870.0, 40.0, 19.0), BOOL;
  @VF(107) : @E(1), @R(320.0, 40.0, 40.0, 19.0), BOOL;
  @VF(108) : @E(vob_Byte4), @R(1190.0, 390.0, 110.0, 19.0);
  @VF(110) : @E(vob_Byte3), @R(1190.0, 300.0, 110.0, 19.0);
  @VF(112) : @E(1), @R(320.0, 230.0, 40.0, 19.0), BOOL;
  @VF(113) : @E(vob_Byte9), @R(1190.0, 850.0, 110.0, 19.0);
  @VF(115) : @E(vob_Byte6), @R(1190.0, 580.0, 110.0, 19.0);
  @VF(117) : @E(4), @R(320.0, 340.0, 40.0, 19.0), BYTE;
  @VF(118) : @E(1), @R(320.0, 60.0, 40.0, 19.0), BOOL;
  @VF(119) : @E(vob_Byte1), @R(1190.0, 110.0, 110.0, 19.0);
  @VF(121) : @E(1), @R(320.0, 780.0, 40.0, 19.0), BOOL;
  @VF(122) : @E(3), @R(320.0, 250.0, 40.0, 19.0), BYTE;
  @VF(123) : @E(1), @R(320.0, 410.0, 40.0, 19.0), BOOL;
  @VF(124) : @E(1), @R(320.0, 130.0, 40.0, 19.0), BOOL;
  @VF(125) : @E(vob_Byte0), @R(1190.0, 20.0, 110.0, 19.0);
  @VF(127) : @E(vob_Byte7), @R(1190.0, 670.0, 110.0, 19.0);
  @C(141) : @F(MID), @R(510.0, 110.0, 100.0, 58.0), INT, @I(@N(IN), @L(9.5)), @I(@N(L), @L(29.5)), @I(@N(P), @L(49.5)), @O(@N(MID), @R(9.5));
  @C(142) : @F(TO_INT), @R(390.0, 130.0, 80.0, 18.0), BOOL, @I(@N(IN), @L(9.5)), @O(@N(TO_INT), @R(9.5));
  @C(143) : @F(TO_INT), @R(390.0, 150.0, 80.0, 18.0), BYTE, @I(@N(IN), @L(9.5)), @O(@N(TO_INT), @R(9.5));
  @C(144) : @F(MID), @R(510.0, 210.0, 100.0, 58.0), INT, @I(@N(IN), @L(9.5)), @I(@N(L), @L(29.5)), @I(@N(P), @L(49.5)), @O(@N(MID), @R(9.5));
  @C(145) : @F(MID), @R(510.0, 760.0, 100.0, 58.0), INT, @I(@N(IN), @L(9.5)), @I(@N(L), @L(29.5)), @I(@N(P), @L(49.5)), @O(@N(MID), @R(9.5));
  @C(146) : @F(TO_INT), @R(390.0, 780.0, 80.0, 18.0), BOOL, @I(@N(IN), @L(9.5)), @O(@N(TO_INT), @R(9.5));
  @C(147) : @F(TO_INT), @R(390.0, 800.0, 80.0, 18.0), BYTE, @I(@N(IN), @L(9.5)), @O(@N(TO_INT), @R(9.5));
  @C(148) : @F(TO_INT), @R(390.0, 40.0, 80.0, 18.0), BOOL, @I(@N(IN), @L(9.5)), @O(@N(TO_INT), @R(9.5));
  @C(149) : @F(TO_INT), @R(390.0, 410.0, 80.0, 18.0), BOOL, @I(@N(IN), @L(9.5)), @O(@N(TO_INT), @R(9.5));
  @C(150) : @F(MID), @R(510.0, 580.0, 100.0, 58.0), INT, @I(@N(IN), @L(9.5)), @I(@N(L), @L(29.5)), @I(@N(P), @L(49.5)), @O(@N(MID), @R(9.5));
  @C(151) : @F(TO_INT), @R(390.0, 600.0, 80.0, 18.0), BOOL, @I(@N(IN), @L(9.5)), @O(@N(TO_INT), @R(9.5));
  @C(152) : @F(TO_INT), @R(390.0, 620.0, 80.0, 18.0), BYTE, @I(@N(IN), @L(9.5)), @O(@N(TO_INT), @R(9.5));
  @C(153) : @F(MID), @R(510.0, 20.0, 100.0, 58.0), INT, @I(@N(IN), @L(9.5)), @I(@N(L), @L(29.5)), @I(@N(P), @L(49.5)), @O(@N(MID), @R(9.5));
  @C(154) : @F(TO_INT), @R(390.0, 500.0, 80.0, 18.0), BOOL, @I(@N(IN), @L(9.5)), @O(@N(TO_INT), @R(9.5));
  @C(155) : @F(MID), @R(510.0, 480.0, 100.0, 58.0), INT, @I(@N(IN), @L(9.5)), @I(@N(L), @L(29.5)), @I(@N(P), @L(49.5)), @O(@N(MID), @R(9.5));
  @C(156) : @F(MID), @R(510.0, 390.0, 100.0, 58.0), INT, @I(@N(IN), @L(9.5)), @I(@N(L), @L(29.5)), @I(@N(P), @L(49.5)), @O(@N(MID), @R(9.5));
  @C(157) : @F(TO_INT), @R(390.0, 430.0, 80.0, 18.0), BYTE, @I(@N(IN), @L(9.5)), @O(@N(TO_INT), @R(9.5));
  @C(158) : @F(TO_INT), @R(390.0, 520.0, 80.0, 18.0), BYTE, @I(@N(IN), @L(9.5)), @O(@N(TO_INT), @R(9.5));
  @C(159) : @F(TO_INT), @R(390.0, 250.0, 80.0, 18.0), BYTE, @I(@N(IN), @L(9.5)), @O(@N(TO_INT), @R(9.5));
  @C(160) : @F(TO_INT), @R(390.0, 60.0, 80.0, 18.0), BOOL, @I(@N(IN), @L(9.5)), @O(@N(TO_INT), @R(9.5));
  @C(161) : @F(MID), @R(510.0, 850.0, 100.0, 58.0), INT, @I(@N(IN), @L(9.5)), @I(@N(L), @L(29.5)), @I(@N(P), @L(49.5)), @O(@N(MID), @R(9.5));
  @C(162) : @F(TO_INT), @R(390.0, 870.0, 80.0, 18.0), BOOL, @I(@N(IN), @L(9.5)), @O(@N(TO_INT), @R(9.5));
  @C(163) : @F(TO_INT), @R(390.0, 890.0, 80.0, 18.0), BYTE, @I(@N(IN), @L(9.5)), @O(@N(TO_INT), @R(9.5));
  @C(164) : @F(MID), @R(510.0, 670.0, 100.0, 58.0), INT, @I(@N(IN), @L(9.5)), @I(@N(L), @L(29.5)), @I(@N(P), @L(49.5)), @O(@N(MID), @R(9.5));
  @C(165) : @F(TO_INT), @R(390.0, 690.0, 80.0, 18.0), BOOL, @I(@N(IN), @L(9.5)), @O(@N(TO_INT), @R(9.5));
  @C(166) : @F(TO_INT), @R(390.0, 710.0, 80.0, 18.0), BYTE, @I(@N(IN), @L(9.5)), @O(@N(TO_INT), @R(9.5));
  @C(167) : @F(MID), @R(510.0, 300.0, 100.0, 58.0), INT, @I(@N(IN), @L(9.5)), @I(@N(L), @L(29.5)), @I(@N(P), @L(49.5)), @O(@N(MID), @R(9.5));
  @C(168) : @F(TO_INT), @R(390.0, 320.0, 80.0, 18.0), BOOL, @I(@N(IN), @L(9.5)), @O(@N(TO_INT), @R(9.5));
  @C(169) : @F(TO_INT), @R(390.0, 230.0, 80.0, 18.0), BOOL, @I(@N(IN), @L(9.5)), @O(@N(TO_INT), @R(9.5));
  @C(170) : @F(TO_INT), @R(390.0, 340.0, 80.0, 18.0), BYTE, @I(@N(IN), @L(9.5)), @O(@N(TO_INT), @R(9.5));
  @C(128) : @FB(FB_lc_ChrToByte7), @R(690.0, 670.0, 200.0, 58.0), @I(@N(vistr_Chr_127), @L(9.5)), @O(@N(vob_Out), @R(9.5));
  @C(140) : @FB(FB_lc_ChrToByte8), @R(690.0, 760.0, 200.0, 58.0), @I(@N(vistr_Chr_127), @L(9.5)), @O(@N(vob_Out), @R(9.5));
  @C(102) : @FB(FB_lc_ChrToByte), @R(690.0, 210.0, 200.0, 58.0), @I(@N(vistr_Chr_127), @L(9.5)), @O(@N(vob_Out), @R(9.5));
  @C(104) : @FB(FB_lc_ChrToByte5), @R(690.0, 480.0, 200.0, 58.0), @I(@N(vistr_Chr_127), @L(9.5)), @O(@N(vob_Out), @R(9.5));
  @C(109) : @FB(FB_lc_ChrToByte4), @R(690.0, 390.0, 200.0, 58.0), @I(@N(vistr_Chr_127), @L(9.5)), @O(@N(vob_Out), @R(9.5));
  @C(111) : @FB(FB_lc_ChrToByte3), @R(690.0, 300.0, 200.0, 58.0), @I(@N(vistr_Chr_127), @L(9.5)), @O(@N(vob_Out), @R(9.5));
  @C(114) : @FB(FB_lc_ChrToByte9), @R(690.0, 850.0, 200.0, 58.0), @I(@N(vistr_Chr_127), @L(9.5)), @O(@N(vob_Out), @R(9.5));
  @C(116) : @FB(FB_lc_ChrToByte6), @R(690.0, 580.0, 200.0, 58.0), @I(@N(vistr_Chr_127), @L(9.5)), @O(@N(vob_Out), @R(9.5));
  @C(120) : @FB(FB_lc_ChrToByte1), @R(690.0, 110.0, 200.0, 58.0), @I(@N(vistr_Chr_127), @L(9.5)), @O(@N(vob_Out), @R(9.5));
  @C(126) : @FB(FB_lc_ChrToByte2), @R(690.0, 20.0, 200.0, 58.0), @I(@N(vistr_Chr_127), @L(9.5)), @O(@N(vob_Out), @R(9.5));
  @CP(184) : 310.0, 29.5;
  @CP(185) : 310.0, 119.5;
  @CP(190) : 310.0, 219.5;
  @CP(193) : 310.0, 309.5;
  @CP(194) : 310.0, 399.5;
  @CP(195) : 310.0, 489.5;
  @CP(196) : 310.0, 589.5;
  @CP(197) : 310.0, 679.5;
  @CP(198) : 310.0, 769.5;

  @G(183) :
     @L(@VF(132).o, @CP(184)),
     @L(@CP(184), @CP(185)),
     @L(@CP(185), @C(141).IN),
     @L(@CP(185), @CP(190)),
     @L(@CP(190), @C(144).IN),
     @L(@CP(190), @CP(193)),
     @L(@CP(193), @CP(194)),
     @L(@CP(194), @CP(195)),
     @L(@CP(195), @CP(196)),
     @L(@CP(196), @CP(197)),
     @L(@CP(197), @CP(198)),
     @L(@CP(198), @C(145).IN),
     @L(@CP(196), @C(150).IN),
     @L(@CP(184), @C(153).IN),
     @L(@CP(195), @C(155).IN),
     @L(@CP(194), @C(156).IN),
     @L(@CP(198), @C(161).IN),
     @L(@CP(197), @C(164).IN),
     @L(@CP(193), @C(167).IN)
    ;
  @G(186) :
     @L(@C(142).TO_INT, @C(141).L)
    ;
  @G(187) :
     @L(@C(143).TO_INT, @C(141).P)
    ;
  @G(188) :
     @L(@VF(124).o, @C(142).IN)
    ;
  @G(189) :
     @L(@VF(130).o, @C(143).IN)
    ;
  @G(191) :
     @L(@C(169).TO_INT, @C(144).L)
    ;
  @G(192) :
     @L(@C(159).TO_INT, @C(144).P)
    ;
  @G(199) :
     @L(@C(146).TO_INT, @C(145).L)
    ;
  @G(200) :
     @L(@C(147).TO_INT, @C(145).P)
    ;
  @G(201) :
     @L(@VF(121).o, @C(146).IN)
    ;
  @G(202) :
     @L(@VF(133).o, @C(147).IN)
    ;
  @G(203) :
     @L(@VF(107).o, @C(148).IN)
    ;
  @G(204) :
     @L(@VF(123).o, @C(149).IN)
    ;
  @G(205) :
     @L(@C(151).TO_INT, @C(150).L)
    ;
  @G(206) :
     @L(@C(152).TO_INT, @C(150).P)
    ;
  @G(207) :
     @L(@VF(136).o, @C(151).IN)
    ;
  @G(208) :
     @L(@VF(105).o, @C(152).IN)
    ;
  @G(209) :
     @L(@C(148).TO_INT, @C(153).L)
    ;
  @G(210) :
     @L(@C(160).TO_INT, @C(153).P)
    ;
  @G(211) :
     @L(@VF(100).o, @C(154).IN)
    ;
  @G(212) :
     @L(@C(154).TO_INT, @C(155).L)
    ;
  @G(213) :
     @L(@C(158).TO_INT, @C(155).P)
    ;
  @G(214) :
     @L(@C(149).TO_INT, @C(156).L)
    ;
  @G(215) :
     @L(@C(157).TO_INT, @C(156).P)
    ;
  @G(216) :
     @L(@VF(137).o, @C(157).IN)
    ;
  @G(217) :
     @L(@VF(138).o, @C(158).IN)
    ;
  @G(218) :
     @L(@VF(122).o, @C(159).IN)
    ;
  @G(219) :
     @L(@VF(118).o, @C(160).IN)
    ;
  @G(220) :
     @L(@C(162).TO_INT, @C(161).L)
    ;
  @G(221) :
     @L(@C(163).TO_INT, @C(161).P)
    ;
  @G(222) :
     @L(@VF(106).o, @C(162).IN)
    ;
  @G(223) :
     @L(@VF(135).o, @C(163).IN)
    ;
  @G(224) :
     @L(@C(165).TO_INT, @C(164).L)
    ;
  @G(225) :
     @L(@C(166).TO_INT, @C(164).P)
    ;
  @G(226) :
     @L(@VF(129).o, @C(165).IN)
    ;
  @G(227) :
     @L(@VF(131).o, @C(166).IN)
    ;
  @G(229) :
     @L(@C(168).TO_INT, @C(167).L)
    ;
  @G(230) :
     @L(@C(170).TO_INT, @C(167).P)
    ;
  @G(231) :
     @L(@VF(134).o, @C(168).IN)
    ;
  @G(233) :
     @L(@VF(112).o, @C(169).IN)
    ;
  @G(234) :
     @L(@VF(117).o, @C(170).IN)
    ;
  @G(1) :
     @L(@C(153).MID, @C(126).vistr_Chr_127)
    ;
  @G(2) :
     @L(@C(141).MID, @C(120).vistr_Chr_127)
    ;
  @G(3) :
     @L(@C(144).MID, @C(102).vistr_Chr_127)
    ;
  @G(4) :
     @L(@C(167).MID, @C(111).vistr_Chr_127)
    ;
  @G(5) :
     @L(@C(156).MID, @C(109).vistr_Chr_127)
    ;
  @G(6) :
     @L(@C(155).MID, @C(104).vistr_Chr_127)
    ;
  @G(7) :
     @L(@C(126).vob_Out, @VF(125).i)
    ;
  @G(8) :
     @L(@C(120).vob_Out, @VF(119).i)
    ;
  @G(9) :
     @L(@C(102).vob_Out, @VF(101).i)
    ;
  @G(10) :
     @L(@C(111).vob_Out, @VF(110).i)
    ;
  @G(11) :
     @L(@C(109).vob_Out, @VF(108).i)
    ;
  @G(12) :
     @L(@C(104).vob_Out, @VF(103).i)
    ;
  @G(13) :
     @L(@C(116).vob_Out, @VF(115).i)
    ;
  @G(14) :
     @L(@C(128).vob_Out, @VF(127).i)
    ;
  @G(15) :
     @L(@C(140).vob_Out, @VF(139).i)
    ;
  @G(16) :
     @L(@C(114).vob_Out, @VF(113).i)
    ;
  @G(17) :
     @L(@C(161).MID, @C(114).vistr_Chr_127)
    ;
  @G(18) :
     @L(@C(145).MID, @C(140).vistr_Chr_127)
    ;
  @G(19) :
     @L(@C(164).MID, @C(128).vistr_Chr_127)
    ;
  @G(20) :
     @L(@C(150).MID, @C(116).vistr_Chr_127)
    ;
END_FUNCTION_BLOCK
END_NAMESPACE

(* ---- FB_lc_TimeToDays_FBD.iecfbd ---- *)
NAMESPACE com.logicals.Basic.Convert
FUNCTION_BLOCK FB_lc_TimeToDays_FBD
  VAR
    UUID_D0B4593F_A5CB_4A31_89F5_7C421E9CAC6A : ForceMrk;
    UUID_95358CAA_7702_4AF4_9B22_BFAB69DBF30F : ForceMrk;
    UUID_9EDBE6A6_63EC_4267_B8F6_98045CA94CD6 : ForceMrk;
  END_VAR
  VAR_INPUT
    vit_In : TIME;
  END_VAR
  VAR_OUTPUT
    vodi_Day : DINT;
    vodi_Hour : DINT;
    vodi_Min : DINT;
    vodi_Sec : DINT;
  END_VAR

  (*

    // Network 1:
    TO_DINT(IN := vit_In, TO_DINT => @C(117).TO_DINT);
    UUID_D0B4593F_A5CB_4A31_89F5_7C421E9CAC6A(IN := @C(117).TO_DINT);
    DIV(IN1 := UUID_D0B4593F_A5CB_4A31_89F5_7C421E9CAC6A.OUT, IN2 := 86400, DIV => (@C(112).DIV, vodi_Day));
    MUL(IN1 := @C(112).DIV, IN2 := 86400, MUL => @C(120).MUL);
    SUB(IN1 := UUID_D0B4593F_A5CB_4A31_89F5_7C421E9CAC6A.OUT, IN2 := @C(120).MUL, SUB => @C(121).SUB);
    UUID_95358CAA_7702_4AF4_9B22_BFAB69DBF30F(IN := @C(121).SUB);
    DIV(IN1 := UUID_95358CAA_7702_4AF4_9B22_BFAB69DBF30F.OUT, IN2 := 3600, DIV => (@C(106).DIV, vodi_Hour));
    MUL(IN1 := @C(106).DIV, IN2 := 3600, MUL => @C(113).MUL);
    SUB(IN1 := UUID_95358CAA_7702_4AF4_9B22_BFAB69DBF30F.OUT, IN2 := @C(113).MUL, SUB => @C(116).SUB);
    UUID_9EDBE6A6_63EC_4267_B8F6_98045CA94CD6(IN := @C(116).SUB);
    DIV(IN1 := UUID_9EDBE6A6_63EC_4267_B8F6_98045CA94CD6.OUT, IN2 := 60, DIV => (@C(104).DIV, vodi_Min));
    MUL(IN1 := @C(104).DIV, IN2 := 60, MUL => @C(115).MUL);
    SUB(IN1 := UUID_9EDBE6A6_63EC_4267_B8F6_98045CA94CD6.OUT, IN2 := @C(115).MUL, SUB => vodi_Sec);

  *)

  @VF(101) : @E(3600), @R(700.0, 210.0, 80.0, 19.0), DINT;
  @VF(102) : @E(86400), @R(370.0, 160.0, 80.0, 19.0), DINT;
  @VF(103) : @E(vodi_Min), @R(1380.0, 240.0, 140.0, 19.0);
  @VF(105) : @E(vodi_Hour), @R(1380.0, 190.0, 140.0, 19.0);
  @VF(107) : @E(vodi_Sec), @R(1380.0, 290.0, 140.0, 19.0);
  @VF(109) : @E(60), @R(1030.0, 260.0, 80.0, 19.0), DINT;
  @VF(110) : @E(vit_In), @R(90.0, 140.0, 110.0, 19.0);
  @VF(111) : @E(vodi_Day), @R(1380.0, 140.0, 140.0, 19.0);
  @C(104) : @F(DIV), @R(1170.0, 240.0, 40.0, 38.0), DINT, @I(@N(IN1), @L(9.5)), @I(@N(IN2), @L(29.5)), @O(@N(DIV), @R(9.5));
  @C(106) : @F(DIV), @R(840.0, 190.0, 40.0, 38.0), DINT, @I(@N(IN1), @L(9.5)), @I(@N(IN2), @L(29.5)), @O(@N(DIV), @R(9.5));
  @C(108) : @F(SUB), @R(1310.0, 290.0, 40.0, 38.0), DINT, @I(@N(IN1), @L(9.5)), @I(@N(IN2), @L(29.5)), @O(@N(SUB), @R(9.5));
  @C(112) : @F(DIV), @R(510.0, 140.0, 40.0, 38.0), DINT, @I(@N(IN1), @L(9.5)), @I(@N(IN2), @L(29.5)), @O(@N(DIV), @R(9.5));
  @C(113) : @F(MUL), @R(920.0, 260.0, 40.0, 38.0), DINT, @I(@N(IN1), @L(9.5)), @I(@N(IN2), @L(29.5)), @O(@N(MUL), @R(9.5));
  @C(114) : @FB(UUID_95358CAA_7702_4AF4_9B22_BFAB69DBF30F), @R(700.0, 190.0, 90.0, 18.0), DINT, @I(@N(IN), @L(9.5)), @O(@N(OUT), @R(9.5));
  @C(115) : @F(MUL), @R(1250.0, 310.0, 40.0, 38.0), DINT, @I(@N(IN1), @L(9.5)), @I(@N(IN2), @L(29.5)), @O(@N(MUL), @R(9.5));
  @C(116) : @F(SUB), @R(980.0, 240.0, 40.0, 38.0), DINT, @I(@N(IN1), @L(9.5)), @I(@N(IN2), @L(29.5)), @O(@N(SUB), @R(9.5));
  @C(117) : @F(TO_DINT), @R(250.0, 140.0, 80.0, 18.0), TIME, @I(@N(IN), @L(9.5)), @O(@N(TO_DINT), @R(9.5));
  @C(118) : @FB(UUID_9EDBE6A6_63EC_4267_B8F6_98045CA94CD6), @R(1030.0, 240.0, 90.0, 18.0), DINT, @I(@N(IN), @L(9.5)), @O(@N(OUT), @R(9.5));
  @C(119) : @FB(UUID_D0B4593F_A5CB_4A31_89F5_7C421E9CAC6A), @R(370.0, 140.0, 90.0, 18.0), DINT, @I(@N(IN), @L(9.5)), @O(@N(OUT), @R(9.5));
  @C(120) : @F(MUL), @R(590.0, 210.0, 40.0, 38.0), DINT, @I(@N(IN1), @L(9.5)), @I(@N(IN2), @L(29.5)), @O(@N(MUL), @R(9.5));
  @C(121) : @F(SUB), @R(650.0, 190.0, 40.0, 38.0), DINT, @I(@N(IN1), @L(9.5)), @I(@N(IN2), @L(29.5)), @O(@N(SUB), @R(9.5));
  @CF(100) : @R(630.0, 50.0, 620.0, 59.0), @T("60s=1min$R$N60min=1h = $a03.600s$R$N24h=1day = 86.400s"), @POU;
  @CP(123) : 1230.0, 249.5;
  @CP(125) : 900.0, 199.5;
  @CP(128) : 570.0, 149.5;
  @CP(130) : 1150.0, 249.5;
  @CP(132) : 1130.0, 269.5;
  @CP(134) : 820.0, 199.5;
  @CP(136) : 800.0, 219.5;
  @CP(139) : 490.0, 149.5;
  @CP(141) : 470.0, 169.5;

  @G(122) :
     @L(@C(104).DIV, @CP(123)),
     @L(@CP(123), @VF(103).i),
     @L(@CP(123), @C(115).IN1)
    ;
  @G(124) :
     @L(@C(106).DIV, @CP(125)),
     @L(@CP(125), @VF(105).i),
     @L(@CP(125), @C(113).IN1)
    ;
  @G(126) :
     @L(@C(108).SUB, @VF(107).i)
    ;
  @G(127) :
     @L(@C(112).DIV, @CP(128)),
     @L(@CP(128), @VF(111).i),
     @L(@CP(128), @C(120).IN1)
    ;
  @G(129) :
     @L(@C(118).OUT, @CP(130)),
     @L(@CP(130), @C(104).IN1),
     @L(@CP(130), @C(108).IN1)
    ;
  @G(131) :
     @L(@VF(109).o, @CP(132)),
     @L(@CP(132), @C(104).IN2),
     @L(@CP(132), @C(115).IN2)
    ;
  @G(133) :
     @L(@C(114).OUT, @CP(134)),
     @L(@CP(134), @C(106).IN1),
     @L(@CP(134), @C(116).IN1)
    ;
  @G(135) :
     @L(@VF(101).o, @CP(136)),
     @L(@CP(136), @C(106).IN2),
     @L(@CP(136), @C(113).IN2)
    ;
  @G(137) :
     @L(@C(115).MUL, @C(108).IN2)
    ;
  @G(138) :
     @L(@C(119).OUT, @CP(139)),
     @L(@CP(139), @C(112).IN1),
     @L(@CP(139), @C(121).IN1)
    ;
  @G(140) :
     @L(@VF(102).o, @CP(141)),
     @L(@CP(141), @C(112).IN2),
     @L(@CP(141), @C(120).IN2)
    ;
  @G(142) :
     @L(@C(121).SUB, @C(114).IN)
    ;
  @G(143) :
     @L(@C(113).MUL, @C(116).IN2)
    ;
  @G(144) :
     @L(@VF(110).o, @C(117).IN)
    ;
  @G(145) :
     @L(@C(116).SUB, @C(118).IN)
    ;
  @G(146) :
     @L(@C(117).TO_DINT, @C(119).IN)
    ;
  @G(147) :
     @L(@C(120).MUL, @C(121).IN2)
    ;
END_FUNCTION_BLOCK
END_NAMESPACE
